(* PLC project Tc2_Standard.WREPLACE Demo, tc3-libraries-kb TwinCAT 3.1 *)
(* stored: creationDateTime 2026-05-11T08:00:00, modificationDateTime 2026-05-11T08:00:00 *)

PROGRAM P_Demo_WREPLACE
  VAR
    sLogLine : WSTRING := "警告 电机异常";  (* 原始中文日志：等级 + 空格 + 消息体 *)
    sNewLevel : WSTRING := "错误";  (* 升级后的等级标识 *)
    sResult : WSTRING;  (* 等级升级后的完整日志 *)
    nReplaceLen : INT := 2;  (* 被替换段字符数 = 2（"警告" 2 个汉字） *)
    nReplacePos : INT := 1;  (* 替换起点 = 第 1 字符 *)
    bUpgrade : BOOL;  (* 触发一次等级升级 *)
  END_VAR

// =============================================================================
// 场景：报警系统判定某条 "警告" 级中文日志在 30 秒内累积 5 次未恢复，需要
//       升级为 "错误" 重发到值班手机。WREPLACE 一行调用把前 2 字 "警告"
//       换成 "错误"，消息体保持不变。
//
// 价值：WREPLACE 按 UCS-2 字符算位置和长度，业务侧看到"前 2 字"就是 2 字。
//       STRING + REPLACE 要传 nReplaceLen = 6（按 UTF-8 字节）才行，错位风险大。
//       另：本函数不是模式匹配替换，要替换所有出现必须配合 WFIND 写循环。
//
// 验证步骤：
//   1. 导入本文件、引用 Tc2_Standard、编译、登录、运行
//   2. 在线 monitor sResult（Unicode 显示）
//   3. 在线写 bUpgrade := TRUE
//   4. 下一周期 sResult = "错误 电机异常"
//   5. 把 sNewLevel 改成 "紧急停机"（4 字）+ 再触发 →
//      sResult = "紧急停机 电机异常"（长度自动变长，验证替换段可不等长）
// =============================================================================

// 入参顺序：(STR1, STR2, L, P) — L 在 P 前，按字符算
IF bUpgrade THEN
    sResult := WREPLACE(sLogLine, sNewLevel, nReplaceLen, nReplacePos);
    bUpgrade := FALSE;
END_IF;
END_PROGRAM
